// LS Electric XG5000 project: 과년66_3
// PLC NewPLC
// module base 0 slot 0: 입출력 모듈:XBC-DR20S (DC 24V 입력 12점, 릴레이 출력 8점)

PROGRAM NewProgram (task: 스캔 프로그램)

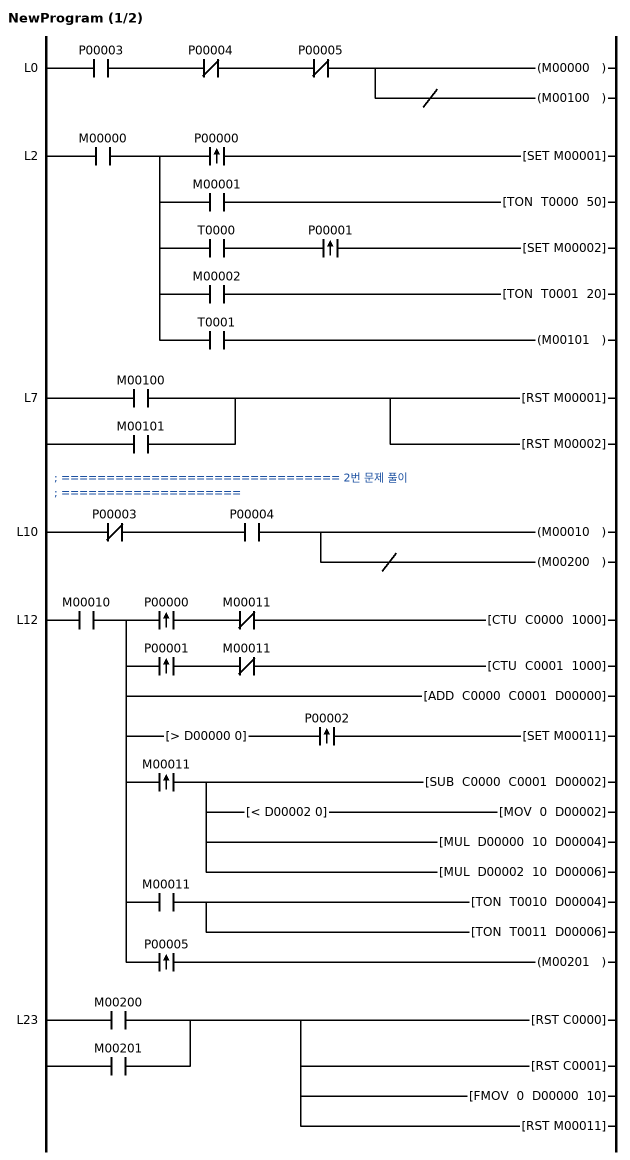
; L0
LOAD      P00003
AND NOT   P00004
AND NOT   P00005
OUT       M00000
NOT
OUT       M00100
; L2
LOAD      M00000
MPUSH
ANDP      P00000
SET       M00001
MLOAD
AND       M00001
TON       T0000 50
MLOAD
AND       T0000
ANDP      P00001
SET       M00002
MLOAD
AND       M00002
TON       T0001 20
MPOP
AND       T0001
OUT       M00101
; L7
LOAD      M00100
OR        M00101
RST       M00001
RST       M00002
// =============================== 2번 문제 풀이 ====================
; L10
LOAD NOT  P00003
AND       P00004
OUT       M00010
NOT
OUT       M00200
; L12
LOAD      M00010
MPUSH
ANDP      P00000
AND NOT   M00011
CTU       C0000 1000
MLOAD
ANDP      P00001
AND NOT   M00011
CTU       C0001 1000
MLOAD
ADD       C0000 C0001 D00000
AND>      D00000 0
ANDP      P00002
SET       M00011
MLOAD
ANDP      M00011
SUB       C0000 C0001 D00002
MPUSH
AND<      D00002 0
MOV       0 D00002
MPOP
MUL       D00000 10 D00004
MUL       D00002 10 D00006
MLOAD
AND       M00011
TON       T0010 D00004
TON       T0011 D00006
MPOP
ANDP      P00005
OUT       M00201
; L23
LOAD      M00200
OR        M00201
RST       C0000
RST       C0001
FMOV      0 D00000 10
RST       M00011

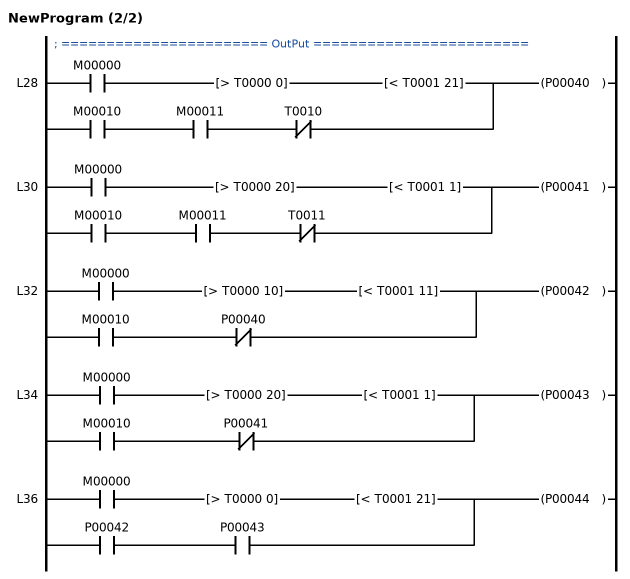
// ======================= OutPut ========================
; L28
LOAD      M00000
AND>      T0000 0
AND<      T0001 21
LOAD      M00010
AND       M00011
AND NOT   T0010
OR LOAD
OUT       P00040
; L30
LOAD      M00000
AND>      T0000 20
AND<      T0001 1
LOAD      M00010
AND       M00011
AND NOT   T0011
OR LOAD
OUT       P00041
; L32
LOAD      M00000
AND>      T0000 10
AND<      T0001 11
LOAD      M00010
AND NOT   P00040
OR LOAD
OUT       P00042
; L34
LOAD      M00000
AND>      T0000 20
AND<      T0001 1
LOAD      M00010
AND NOT   P00041
OR LOAD
OUT       P00043
; L36
LOAD      M00000
AND>      T0000 0
AND<      T0001 21
LOAD      P00042
AND       P00043
OR LOAD
OUT       P00044